// TIA Portal V15.1 export
// export: Created 2024-06-21T08:41:24.4997304Z, ExportSetting WithDefaults, DisplayName Totally Integrated Automation Portal, DisplayVersion V15.1 Update 5, DisplayName TIA Portal Openness, DisplayVersion V15.1 Update 5, DisplayName SINAMICS Startdrive Advanced, DisplayVersion V15.1, DisplayName G130, G150, S120, S150, SINAMICS MV, S210, DisplayVersion V15.1, DisplayName G110M, G120, G120C, G120D, G120P, DisplayVersion V15.1, DisplayName STEP 7 Professional, DisplayVersion V15.1 Update 5, DisplayName STEP 7 Safety, DisplayVersion V15.1, DisplayName WinCC Professional, DisplayVersion V15.1 Update 5, DisplayName SIMATIC Visualization Architect, DisplayVersion V15.1
FUNCTION "209230ZS01Passiv" : Void   // FC423, FBD
TITLE = 209230ZS01Passiv
{ S7_Optimized_Access := 'FALSE' }
AUTHOR : VCC
NAME : LocFunc
VERSION : 0.1
// stored: AutoNumber false, IsIECCheckEnabled false, SetENOAutomatically False, UDAEnableTagReadback false
   VAR_OUTPUT
      O_AlarmA : Bool;   // Alarm A
      O_AlarmB : Bool;   // Alarm B
      O_AlarmC : Bool;   // Alarm C
      O_AlarmD : Bool;   // Alarm D
      O_AlarmABCondition : Bool;   // Alarms resetable
      H_IAnim : Word;   // Icon Animation
   END_VAR
   VAR_TEMP
      TEMP0 : Bool;
   END_VAR
BEGIN

REGION Network 1: **** --------------------- ET200sp I/O --------------------- ****
END_REGION

REGION Network 2: **** 2.2 - Alarms - Alarm Generation **** 209230AS10JX60IF6600 - ET200sp I/O - Safety Card IF6600
   // Passivation alarm - ET200sp I/O - Safety Card IF6600
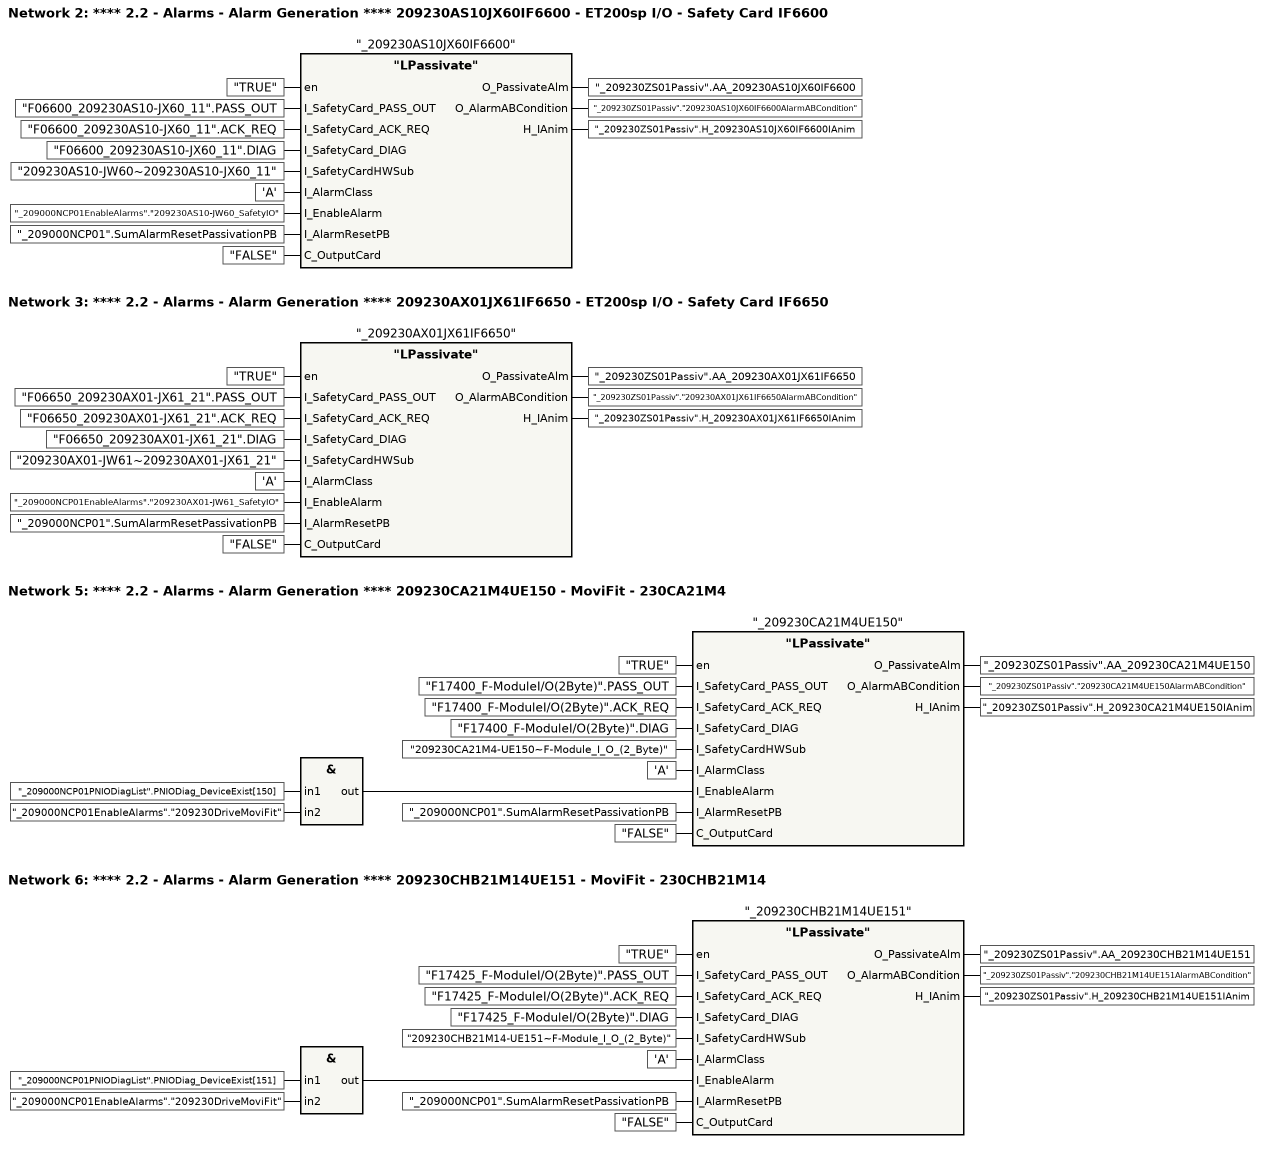
   IF "TRUE" THEN
       "_209230AS10JX60IF6600"(I_SafetyCard_PASS_OUT := "F06600_209230AS10-JX60_11".PASS_OUT,   // "LPassivate"
                               I_SafetyCard_ACK_REQ := "F06600_209230AS10-JX60_11".ACK_REQ,
                               I_SafetyCard_DIAG := "F06600_209230AS10-JX60_11".DIAG,
                               I_SafetyCardHWSub := "209230AS10-JW60~209230AS10-JX60_11",
                               I_AlarmClass := 'A',
                               I_EnableAlarm := "_209000NCP01EnableAlarms"."209230AS10-JW60_SafetyIO",
                               I_AlarmResetPB := "_209000NCP01".SumAlarmResetPassivationPB,
                               C_OutputCard := "FALSE",
                               O_PassivateAlm => "_209230ZS01Passiv".AA_209230AS10JX60IF6600,
                               O_AlarmABCondition => "_209230ZS01Passiv"."209230AS10JX60IF6600AlarmABCondition",
                               H_IAnim => "_209230ZS01Passiv".H_209230AS10JX60IF6600IAnim);
   END_IF;
END_REGION

REGION Network 3: **** 2.2 - Alarms - Alarm Generation **** 209230AX01JX61IF6650 - ET200sp I/O - Safety Card IF6650
   // Passivation alarm - ET200sp I/O - Safety Card IF6650
   IF "TRUE" THEN
       "_209230AX01JX61IF6650"(I_SafetyCard_PASS_OUT := "F06650_209230AX01-JX61_21".PASS_OUT,   // "LPassivate"
                               I_SafetyCard_ACK_REQ := "F06650_209230AX01-JX61_21".ACK_REQ,
                               I_SafetyCard_DIAG := "F06650_209230AX01-JX61_21".DIAG,
                               I_SafetyCardHWSub := "209230AX01-JW61~209230AX01-JX61_21",
                               I_AlarmClass := 'A',
                               I_EnableAlarm := "_209000NCP01EnableAlarms"."209230AX01-JW61_SafetyIO",
                               I_AlarmResetPB := "_209000NCP01".SumAlarmResetPassivationPB,
                               C_OutputCard := "FALSE",
                               O_PassivateAlm => "_209230ZS01Passiv".AA_209230AX01JX61IF6650,
                               O_AlarmABCondition => "_209230ZS01Passiv"."209230AX01JX61IF6650AlarmABCondition",
                               H_IAnim => "_209230ZS01Passiv".H_209230AX01JX61IF6650IAnim);
   END_IF;
END_REGION

REGION Network 4: **** --------------------- Drive --------------------- ****
END_REGION

REGION Network 5: **** 2.2 - Alarms - Alarm Generation **** 209230CA21M4UE150 - MoviFit - 230CA21M4
   // Passivation alarm - MoviFit - 230CA21M4
   IF "TRUE" THEN
       "_209230CA21M4UE150"(I_SafetyCard_PASS_OUT := "F17400_F-ModuleI/O(2Byte)".PASS_OUT,   // "LPassivate"
                            I_SafetyCard_ACK_REQ := "F17400_F-ModuleI/O(2Byte)".ACK_REQ,
                            I_SafetyCard_DIAG := "F17400_F-ModuleI/O(2Byte)".DIAG,
                            I_SafetyCardHWSub := "209230CA21M4-UE150~F-Module_I_O_(2_Byte)",
                            I_AlarmClass := 'A',
                            I_EnableAlarm := "_209000NCP01PNIODiagList".PNIODiag_DeviceExist[150] AND "_209000NCP01EnableAlarms"."209230DriveMoviFit",
                            I_AlarmResetPB := "_209000NCP01".SumAlarmResetPassivationPB,
                            C_OutputCard := "FALSE",
                            O_PassivateAlm => "_209230ZS01Passiv".AA_209230CA21M4UE150,
                            O_AlarmABCondition => "_209230ZS01Passiv"."209230CA21M4UE150AlarmABCondition",
                            H_IAnim => "_209230ZS01Passiv".H_209230CA21M4UE150IAnim);
   END_IF;
END_REGION

REGION Network 6: **** 2.2 - Alarms - Alarm Generation **** 209230CHB21M14UE151 - MoviFit - 230CHB21M14
   // Passivation alarm - MoviFit - 230CHB21M14
   IF "TRUE" THEN
       "_209230CHB21M14UE151"(I_SafetyCard_PASS_OUT := "F17425_F-ModuleI/O(2Byte)".PASS_OUT,   // "LPassivate"
                              I_SafetyCard_ACK_REQ := "F17425_F-ModuleI/O(2Byte)".ACK_REQ,
                              I_SafetyCard_DIAG := "F17425_F-ModuleI/O(2Byte)".DIAG,
                              I_SafetyCardHWSub := "209230CHB21M14-UE151~F-Module_I_O_(2_Byte)",
                              I_AlarmClass := 'A',
                              I_EnableAlarm := "_209000NCP01PNIODiagList".PNIODiag_DeviceExist[151] AND "_209000NCP01EnableAlarms"."209230DriveMoviFit",
                              I_AlarmResetPB := "_209000NCP01".SumAlarmResetPassivationPB,
                              C_OutputCard := "FALSE",
                              O_PassivateAlm => "_209230ZS01Passiv".AA_209230CHB21M14UE151,
                              O_AlarmABCondition => "_209230ZS01Passiv"."209230CHB21M14UE151AlarmABCondition",
                              H_IAnim => "_209230ZS01Passiv".H_209230CHB21M14UE151IAnim);
   END_IF;
END_REGION

REGION Network 7: **** 2.2 - Alarms - Alarm Generation **** 209230CHB22M14UE152 - MoviFit - 230CHB22M14
   // Passivation alarm - MoviFit - 230CHB22M14
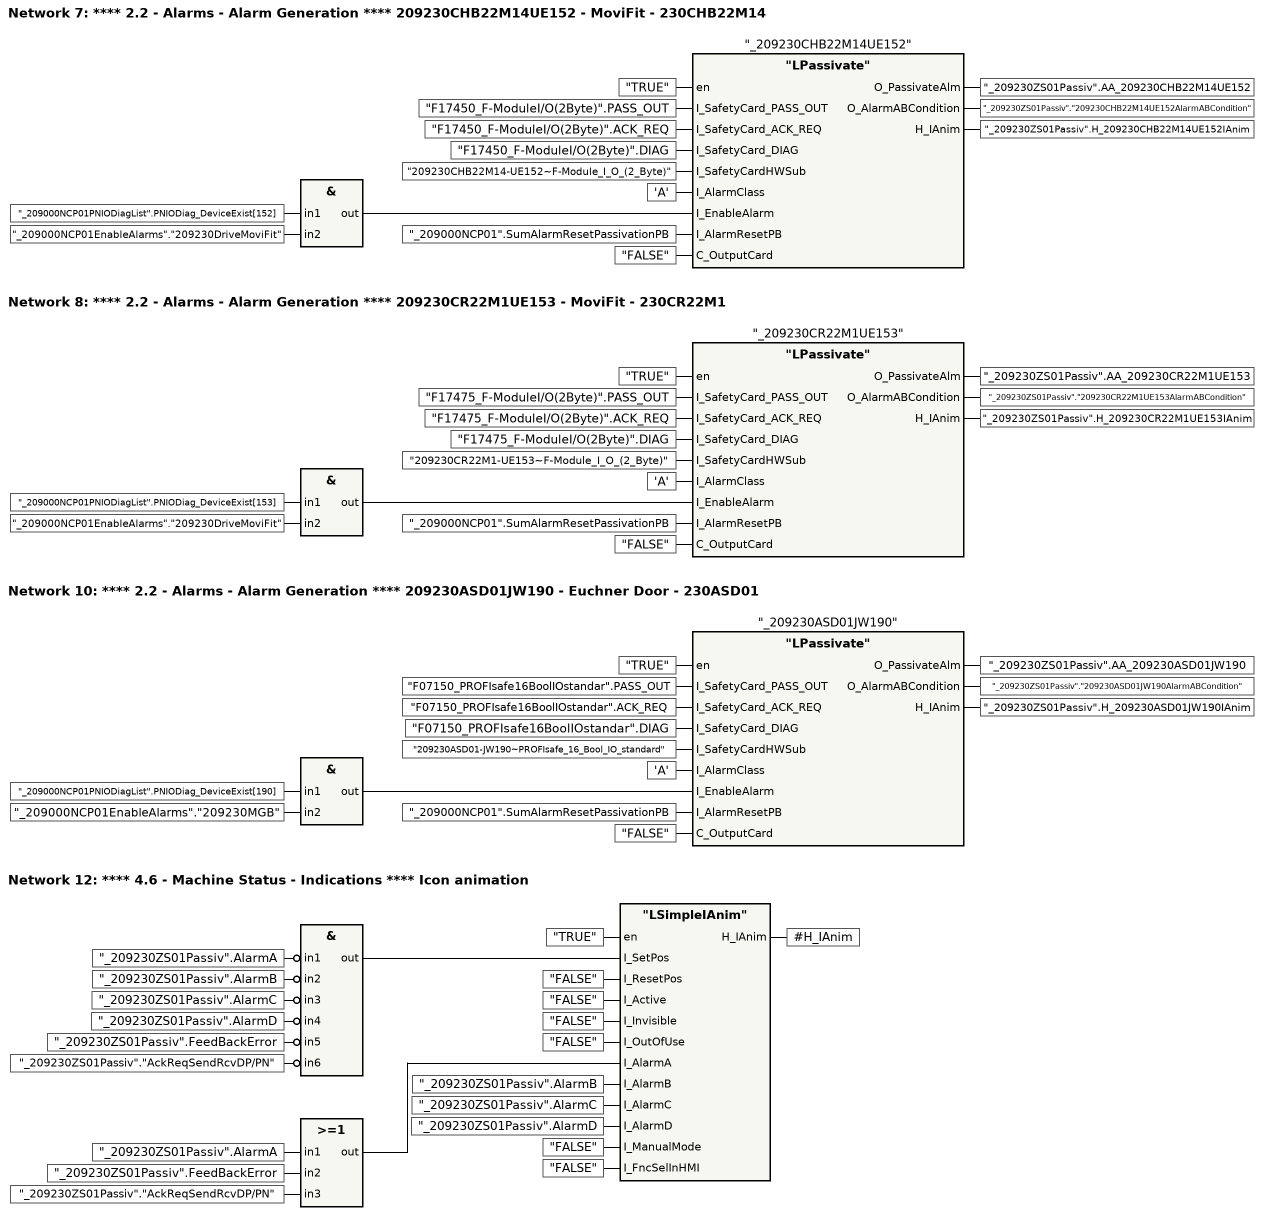
   IF "TRUE" THEN
       "_209230CHB22M14UE152"(I_SafetyCard_PASS_OUT := "F17450_F-ModuleI/O(2Byte)".PASS_OUT,   // "LPassivate"
                              I_SafetyCard_ACK_REQ := "F17450_F-ModuleI/O(2Byte)".ACK_REQ,
                              I_SafetyCard_DIAG := "F17450_F-ModuleI/O(2Byte)".DIAG,
                              I_SafetyCardHWSub := "209230CHB22M14-UE152~F-Module_I_O_(2_Byte)",
                              I_AlarmClass := 'A',
                              I_EnableAlarm := "_209000NCP01PNIODiagList".PNIODiag_DeviceExist[152] AND "_209000NCP01EnableAlarms"."209230DriveMoviFit",
                              I_AlarmResetPB := "_209000NCP01".SumAlarmResetPassivationPB,
                              C_OutputCard := "FALSE",
                              O_PassivateAlm => "_209230ZS01Passiv".AA_209230CHB22M14UE152,
                              O_AlarmABCondition => "_209230ZS01Passiv"."209230CHB22M14UE152AlarmABCondition",
                              H_IAnim => "_209230ZS01Passiv".H_209230CHB22M14UE152IAnim);
   END_IF;
END_REGION

REGION Network 8: **** 2.2 - Alarms - Alarm Generation **** 209230CR22M1UE153 - MoviFit - 230CR22M1
   // Passivation alarm - MoviFit - 230CR22M1
   IF "TRUE" THEN
       "_209230CR22M1UE153"(I_SafetyCard_PASS_OUT := "F17475_F-ModuleI/O(2Byte)".PASS_OUT,   // "LPassivate"
                            I_SafetyCard_ACK_REQ := "F17475_F-ModuleI/O(2Byte)".ACK_REQ,
                            I_SafetyCard_DIAG := "F17475_F-ModuleI/O(2Byte)".DIAG,
                            I_SafetyCardHWSub := "209230CR22M1-UE153~F-Module_I_O_(2_Byte)",
                            I_AlarmClass := 'A',
                            I_EnableAlarm := "_209000NCP01PNIODiagList".PNIODiag_DeviceExist[153] AND "_209000NCP01EnableAlarms"."209230DriveMoviFit",
                            I_AlarmResetPB := "_209000NCP01".SumAlarmResetPassivationPB,
                            C_OutputCard := "FALSE",
                            O_PassivateAlm => "_209230ZS01Passiv".AA_209230CR22M1UE153,
                            O_AlarmABCondition => "_209230ZS01Passiv"."209230CR22M1UE153AlarmABCondition",
                            H_IAnim => "_209230ZS01Passiv".H_209230CR22M1UE153IAnim);
   END_IF;
END_REGION

REGION Network 9: **** --------------------- Euchner Door --------------------- ****
END_REGION

REGION Network 10: **** 2.2 - Alarms - Alarm Generation **** 209230ASD01JW190 - Euchner Door - 230ASD01
   // Passivation alarm - Euchner Door - 230ASD01
   IF "TRUE" THEN
       "_209230ASD01JW190"(I_SafetyCard_PASS_OUT := "F07150_PROFIsafe16BoolIOstandar".PASS_OUT,   // "LPassivate"
                           I_SafetyCard_ACK_REQ := "F07150_PROFIsafe16BoolIOstandar".ACK_REQ,
                           I_SafetyCard_DIAG := "F07150_PROFIsafe16BoolIOstandar".DIAG,
                           I_SafetyCardHWSub := "209230ASD01-JW190~PROFIsafe_16_Bool_IO_standard",
                           I_AlarmClass := 'A',
                           I_EnableAlarm := "_209000NCP01PNIODiagList".PNIODiag_DeviceExist[190] AND "_209000NCP01EnableAlarms"."209230MGB",
                           I_AlarmResetPB := "_209000NCP01".SumAlarmResetPassivationPB,
                           C_OutputCard := "FALSE",
                           O_PassivateAlm => "_209230ZS01Passiv".AA_209230ASD01JW190,
                           O_AlarmABCondition => "_209230ZS01Passiv"."209230ASD01JW190AlarmABCondition",
                           H_IAnim => "_209230ZS01Passiv".H_209230ASD01JW190IAnim);
   END_IF;
END_REGION

REGION Network 11: **** -------------------------------------------------- ****
END_REGION

REGION Network 12: **** 4.6 - Machine Status - Indications **** Icon animation
   // Icon animation
   IF "TRUE" THEN
       "LSimpleIAnim"(I_SetPos := NOT "_209230ZS01Passiv".AlarmA AND NOT "_209230ZS01Passiv".AlarmB AND NOT "_209230ZS01Passiv".AlarmC AND NOT "_209230ZS01Passiv".AlarmD AND NOT "_209230ZS01Passiv".FeedBackError AND NOT "_209230ZS01Passiv"."AckReqSendRcvDP/PN",
                      I_ResetPos := "FALSE",
                      I_Active := "FALSE",
                      I_Invisible := "FALSE",
                      I_OutOfUse := "FALSE",
                      I_AlarmA := "_209230ZS01Passiv".AlarmA OR "_209230ZS01Passiv".FeedBackError OR "_209230ZS01Passiv"."AckReqSendRcvDP/PN",
                      I_AlarmB := "_209230ZS01Passiv".AlarmB,
                      I_AlarmC := "_209230ZS01Passiv".AlarmC,
                      I_AlarmD := "_209230ZS01Passiv".AlarmD,
                      I_ManualMode := "FALSE",
                      I_FncSelInHMI := "FALSE",
                      H_IAnim => #H_IAnim);
   END_IF;
END_REGION

REGION Network 13: **** 4.6 - Machine status - Indications **** Animation
   // Animation
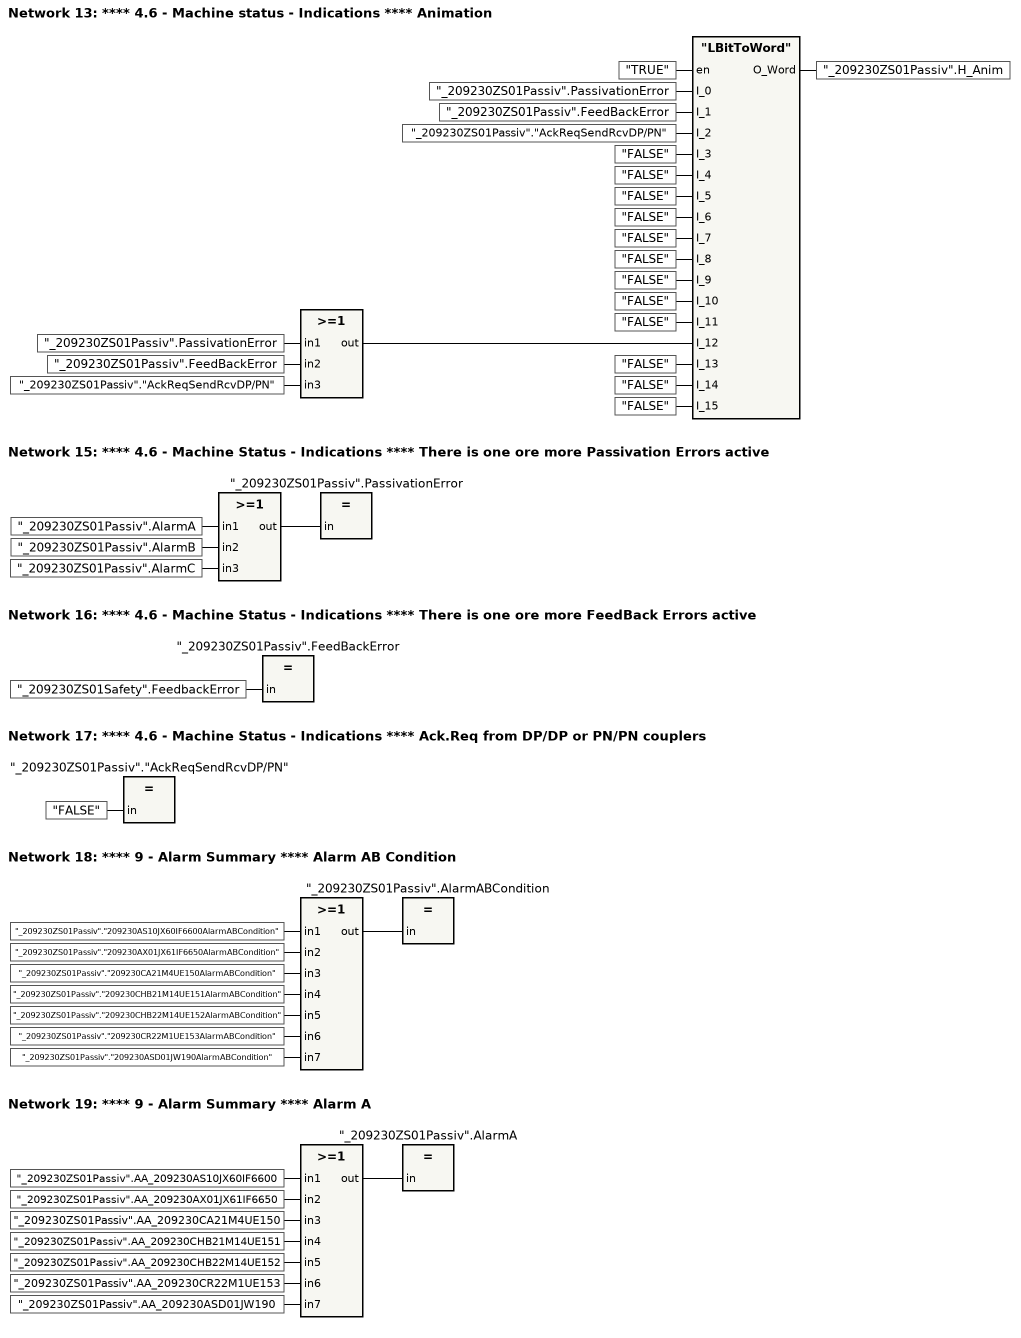
   IF "TRUE" THEN
       "LBitToWord"(I_0 := "_209230ZS01Passiv".PassivationError,
                    I_1 := "_209230ZS01Passiv".FeedBackError,
                    I_2 := "_209230ZS01Passiv"."AckReqSendRcvDP/PN",
                    I_3 := "FALSE",
                    I_4 := "FALSE",
                    I_5 := "FALSE",
                    I_6 := "FALSE",
                    I_7 := "FALSE",
                    I_8 := "FALSE",
                    I_9 := "FALSE",
                    I_10 := "FALSE",
                    I_11 := "FALSE",
                    I_12 := "_209230ZS01Passiv".PassivationError OR "_209230ZS01Passiv".FeedBackError OR "_209230ZS01Passiv"."AckReqSendRcvDP/PN",
                    I_13 := "FALSE",
                    I_14 := "FALSE",
                    I_15 := "FALSE",
                    O_Word => "_209230ZS01Passiv".H_Anim);
   END_IF;
END_REGION

NETWORK
TITLE = **** 4.6 - Machine Status - Indications **** Animation DB number
// DB number
      OPN   "_209230ZS01Passiv";
      L     DBNO;
      T     "_209230ZS01Passiv".H_DBnr;

REGION Network 15: **** 4.6 - Machine Status - Indications **** There is one ore more Passivation Errors active
   // There is one ore more Passivation Errors active
   "_209230ZS01Passiv".PassivationError := "_209230ZS01Passiv".AlarmA OR "_209230ZS01Passiv".AlarmB OR "_209230ZS01Passiv".AlarmC;
END_REGION

REGION Network 16: **** 4.6 - Machine Status - Indications **** There is one ore more FeedBack Errors active
   // There is one ore more FeedBack Errors active
   "_209230ZS01Passiv".FeedBackError := "_209230ZS01Safety".FeedbackError;
END_REGION

REGION Network 17: **** 4.6 - Machine Status - Indications **** Ack.Req from DP/DP or PN/PN couplers
   // Ack.Req from DP/DP or PN/PN couplers
   "_209230ZS01Passiv"."AckReqSendRcvDP/PN" := "FALSE";
END_REGION

REGION Network 18: **** 9 - Alarm Summary **** Alarm AB Condition
   // Alarm AB condition
   "_209230ZS01Passiv".AlarmABCondition := "_209230ZS01Passiv"."209230AS10JX60IF6600AlarmABCondition" OR "_209230ZS01Passiv"."209230AX01JX61IF6650AlarmABCondition" OR "_209230ZS01Passiv"."209230CA21M4UE150AlarmABCondition" OR "_209230ZS01Passiv"."209230CHB21M14UE151AlarmABCondition" OR "_209230ZS01Passiv"."209230CHB22M14UE152AlarmABCondition" OR "_209230ZS01Passiv"."209230CR22M1UE153AlarmABCondition" OR "_209230ZS01Passiv"."209230ASD01JW190AlarmABCondition";
END_REGION

REGION Network 19: **** 9 - Alarm Summary **** Alarm A
   // Summary of alarms A
   "_209230ZS01Passiv".AlarmA := "_209230ZS01Passiv".AA_209230AS10JX60IF6600 OR "_209230ZS01Passiv".AA_209230AX01JX61IF6650 OR "_209230ZS01Passiv".AA_209230CA21M4UE150 OR "_209230ZS01Passiv".AA_209230CHB21M14UE151 OR "_209230ZS01Passiv".AA_209230CHB22M14UE152 OR "_209230ZS01Passiv".AA_209230CR22M1UE153 OR "_209230ZS01Passiv".AA_209230ASD01JW190;
END_REGION

REGION Network 20: **** 9 - Alarm Summary **** Alarm B
   // Summary of alarms B
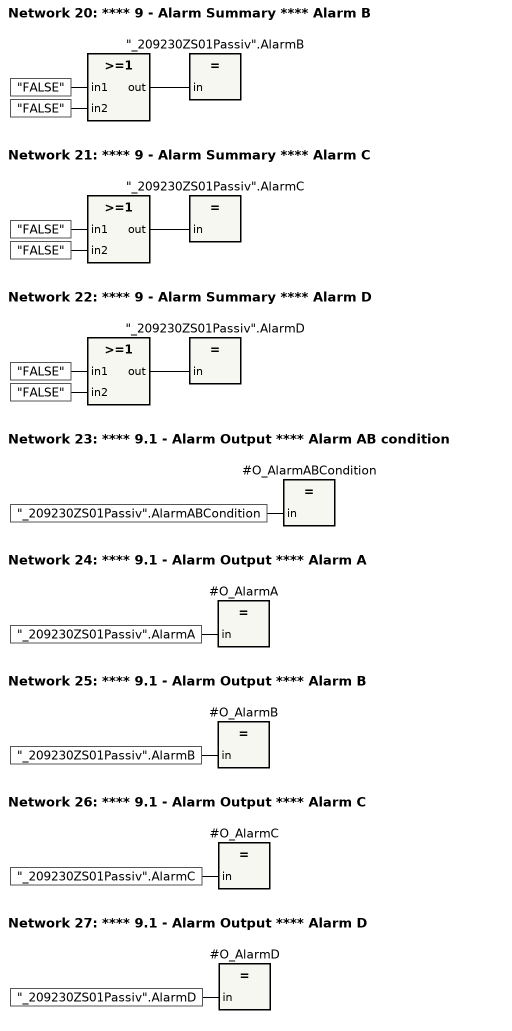
   "_209230ZS01Passiv".AlarmB := "FALSE" OR "FALSE";
END_REGION

REGION Network 21: **** 9 - Alarm Summary **** Alarm C
   // Summary of alarms C
   "_209230ZS01Passiv".AlarmC := "FALSE" OR "FALSE";
END_REGION

REGION Network 22: **** 9 - Alarm Summary **** Alarm D
   // Summary of alarms D
   "_209230ZS01Passiv".AlarmD := "FALSE" OR "FALSE";
END_REGION

REGION Network 23: **** 9.1 - Alarm Output **** Alarm AB condition
   // Alarm AB condition
   #O_AlarmABCondition := "_209230ZS01Passiv".AlarmABCondition;
END_REGION

REGION Network 24: **** 9.1 - Alarm Output **** Alarm A
   // Output Alarm A
   #O_AlarmA := "_209230ZS01Passiv".AlarmA;
END_REGION

REGION Network 25: **** 9.1 - Alarm Output **** Alarm B
   // Output Alarm B
   #O_AlarmB := "_209230ZS01Passiv".AlarmB;
END_REGION

REGION Network 26: **** 9.1 - Alarm Output **** Alarm C
   // Output Alarm C
   #O_AlarmC := "_209230ZS01Passiv".AlarmC;
END_REGION

REGION Network 27: **** 9.1 - Alarm Output **** Alarm D
   // Output Alarm D
   #O_AlarmD := "_209230ZS01Passiv".AlarmD;
END_REGION

REGION Network 28: **** 9.2 - Alarm DWord**** Alarm To DWord
   // Alarm Word
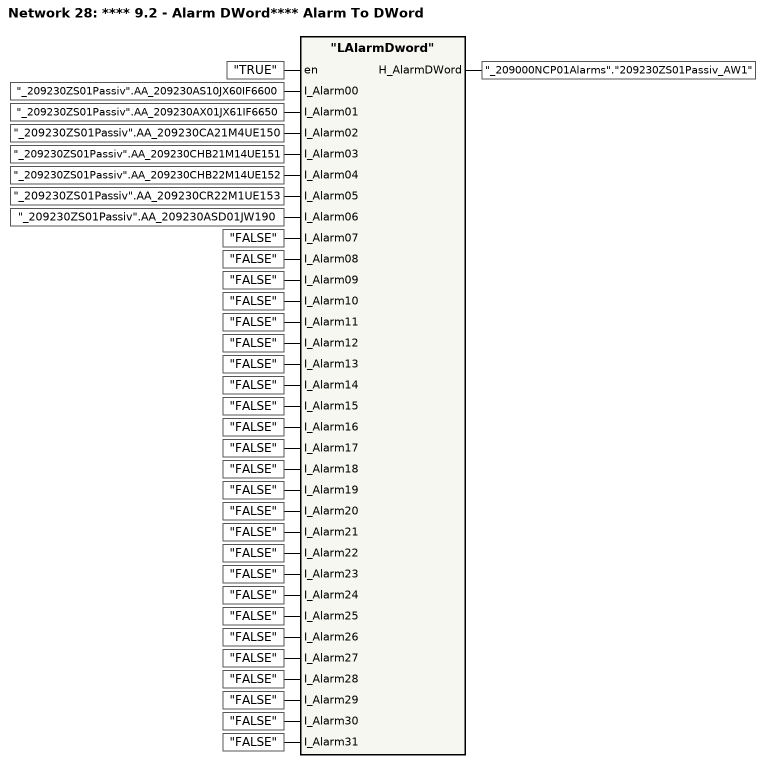
   IF "TRUE" THEN
       "LAlarmDword"(I_Alarm00 := "_209230ZS01Passiv".AA_209230AS10JX60IF6600,
                     I_Alarm01 := "_209230ZS01Passiv".AA_209230AX01JX61IF6650,
                     I_Alarm02 := "_209230ZS01Passiv".AA_209230CA21M4UE150,
                     I_Alarm03 := "_209230ZS01Passiv".AA_209230CHB21M14UE151,
                     I_Alarm04 := "_209230ZS01Passiv".AA_209230CHB22M14UE152,
                     I_Alarm05 := "_209230ZS01Passiv".AA_209230CR22M1UE153,
                     I_Alarm06 := "_209230ZS01Passiv".AA_209230ASD01JW190,
                     I_Alarm07 := "FALSE",
                     I_Alarm08 := "FALSE",
                     I_Alarm09 := "FALSE",
                     I_Alarm10 := "FALSE",
                     I_Alarm11 := "FALSE",
                     I_Alarm12 := "FALSE",
                     I_Alarm13 := "FALSE",
                     I_Alarm14 := "FALSE",
                     I_Alarm15 := "FALSE",
                     I_Alarm16 := "FALSE",
                     I_Alarm17 := "FALSE",
                     I_Alarm18 := "FALSE",
                     I_Alarm19 := "FALSE",
                     I_Alarm20 := "FALSE",
                     I_Alarm21 := "FALSE",
                     I_Alarm22 := "FALSE",
                     I_Alarm23 := "FALSE",
                     I_Alarm24 := "FALSE",
                     I_Alarm25 := "FALSE",
                     I_Alarm26 := "FALSE",
                     I_Alarm27 := "FALSE",
                     I_Alarm28 := "FALSE",
                     I_Alarm29 := "FALSE",
                     I_Alarm30 := "FALSE",
                     I_Alarm31 := "FALSE",
                     H_AlarmDWord => "_209000NCP01Alarms"."209230ZS01Passiv_AW1");
   END_IF;
END_REGION
END_FUNCTION
